INTERFACE ITF_ControlElement5 EXTENDS ITF_BaseControlElement

END_INTERFACE

(* stored: Version 1.1.0.1, ProductVersion 3.1.4024.15
   Itf ITF_ControlElement5: Id {082681d3-8970-4360-885a-57828c59c68f} *)
